(* Logix 5000 project; controller Sistec_test_serial_compact vendor 1 type 14 code 222 rev 36.11; software revision 36.00 *)

TASK MainTask (continuous, watchdog 500 ms) : MainProgram
TASK SafetyTask (periodic, rate 20 ms, priority 10, watchdog 20 ms, safety) : SafetyProgram

MODULES
   Local : vendor 1 type 14 code 222 (5069 0, rev 36.11)
      Sortides : vendor 1 type 7 code 393 (5069 1, rev 3.12, StandardDataDriven RPI 5 ms)
      Entrades : vendor 1 type 7 code 391 (5069 2, rev 2.13, StandardDataDriven RPI 5 ms)
      Serial : vendor 1 type 12 code 320 (5069 4, rev 2.12, StandardDataDriven RPI 80 ms)
      Entrades_analogiques : vendor 1 type 115 code 314 (5069 3, rev 2.12, StandardDataDriven RPI 100 ms)
END_MODULES

VAR_GLOBAL   (* controller tags *)
   Serial_data_compact : INT[10] := ([0] := 10, [1] := 2, [2] := 3, [3] := 4, [4] := 4, [5] := 4, [6] := 5, [7] := 6, [8] := 7, [9] := 8); {produced}
END_VAR

PROGRAM MainProgram   (* main routine MainRoutine *)

ROUTINE MainRoutine   (* ladder *)
   0 (stored rung type 13): ;
END_ROUTINE
END_PROGRAM

PROGRAM SafetyProgram   (* main routine MainRoutine, safety *)

ROUTINE MainRoutine   (* ladder *)
END_ROUTINE
END_PROGRAM
